FUNCTION_BLOCK MQTT_PUBLISHER
  {SET_ATTRIBUTE(OpcUa, POINT.ENDPOINT)}
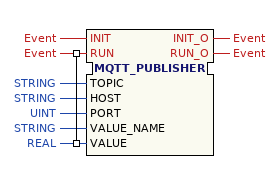
  EVENT_INPUT
    INIT;
    RUN WITH VALUE;
  END_EVENT
  EVENT_OUTPUT
    INIT_O;
    RUN_O;
  END_EVENT
  VAR_INPUT
    TOPIC : STRING; {SET_ATTRIBUTE(OpcUa, Constant)}
    HOST : STRING; {SET_ATTRIBUTE(OpcUa, Constant)}
    PORT : UINT; {SET_ATTRIBUTE(OpcUa, Constant)}
    VALUE_NAME : STRING; {SET_ATTRIBUTE(OpcUa, Constant)}
    VALUE : REAL; {SET_ATTRIBUTE(OpcUa, Variable)}
  END_VAR
END_FUNCTION_BLOCK
